// TIA Portal V20 export
// export: Created 2025-12-01T14:57:22.6291622Z, ExportSetting None, DisplayName Totally Integrated Automation Portal, DisplayVersion V20 Update 3, DisplayName TIA Portal Openness, DisplayVersion V20 Update 3, DisplayName TIA Portal Version Control Interface, DisplayVersion V20 Update 3, DisplayName STEP 7 Professional, DisplayVersion V20 Update 3, DisplayName STEP 7 Safety, DisplayVersion V20 Update 2, DisplayName WinCC Basic/Comfort/Advanced, DisplayVersion V20 Update 3, DisplayName WinCC Professional, DisplayVersion V20 Update 3, DisplayName WinCC Unified, DisplayVersion V20 Update 3
FUNCTION "FC1_Llamadas_CCPIF" : Void   // FC1, LAD
{ S7_Optimized_Access := 'FALSE' }
// stored: AutoNumber false, SetENOAutomatically false
   VAR_TEMP
      FinReset : Bool;
      Luminoso_Verde : Bool;
      Luminoso_Rojo : Bool;
      Luminoso_Naranja : Bool;
   END_VAR
BEGIN

REGION Network 1: Final de Reset
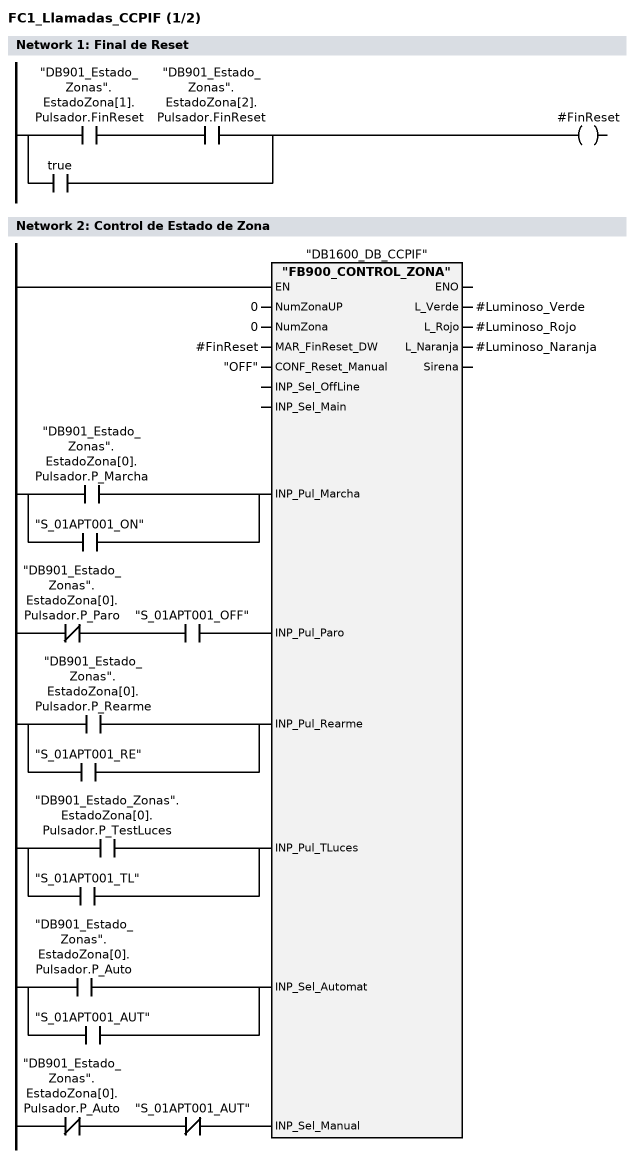
   RUNG wire#powerrail
      Contact( "DB901_Estado_Zonas".EstadoZona[1].Pulsador.FinReset )
      Contact( "DB901_Estado_Zonas".EstadoZona[2].Pulsador.FinReset )
      wire#w1
      Coil( #FinReset )
   END_RUNG
   RUNG wire#powerrail
      Contact( true )
   END_RUNG wire#w1
   // the same network as SCL:
   #FinReset := ("DB901_Estado_Zonas".EstadoZona[1].Pulsador.FinReset AND "DB901_Estado_Zonas".EstadoZona[2].Pulsador.FinReset) OR true;
END_REGION

REGION Network 2: Control de Estado de Zona
   RUNG wire#powerrail
      "DB1600_DB_CCPIF"(INP_Pul_Marcha := wire#w1, INP_Pul_Paro := wire#w2, INP_Pul_Rearme := wire#w3, INP_Pul_TLuces := wire#w4, INP_Sel_Automat := wire#w5, INP_Sel_Manual := wire#w6, NumZonaUP := 0, NumZona := 0, MAR_FinReset_DW := #FinReset, CONF_Reset_Manual := "OFF", INP_Sel_OffLine :=, INP_Sel_Main :=, L_Verde => #Luminoso_Verde, L_Rojo => #Luminoso_Rojo, L_Naranja => #Luminoso_Naranja, Sirena =>)
   END_RUNG
   RUNG wire#powerrail
      Contact( "DB901_Estado_Zonas".EstadoZona[0].Pulsador.P_Marcha )
   END_RUNG wire#w1
   RUNG wire#powerrail
      Contact( "S_01APT001_ON" )
   END_RUNG wire#w1
   RUNG wire#powerrail
      I_Contact( "DB901_Estado_Zonas".EstadoZona[0].Pulsador.P_Paro )
      Contact( "S_01APT001_OFF" )
   END_RUNG wire#w2
   RUNG wire#powerrail
      Contact( "DB901_Estado_Zonas".EstadoZona[0].Pulsador.P_Rearme )
   END_RUNG wire#w3
   RUNG wire#powerrail
      Contact( "S_01APT001_RE" )
   END_RUNG wire#w3
   RUNG wire#powerrail
      Contact( "DB901_Estado_Zonas".EstadoZona[0].Pulsador.P_TestLuces )
   END_RUNG wire#w4
   RUNG wire#powerrail
      Contact( "S_01APT001_TL" )
   END_RUNG wire#w4
   RUNG wire#powerrail
      Contact( "DB901_Estado_Zonas".EstadoZona[0].Pulsador.P_Auto )
   END_RUNG wire#w5
   RUNG wire#powerrail
      Contact( "S_01APT001_AUT" )
   END_RUNG wire#w5
   RUNG wire#powerrail
      I_Contact( "DB901_Estado_Zonas".EstadoZona[0].Pulsador.P_Auto )
      I_Contact( "S_01APT001_AUT" )
   END_RUNG wire#w6
   // the same network as SCL:
   "DB1600_DB_CCPIF"(NumZonaUP := 0,   // "FB900_CONTROL_ZONA"
                     NumZona := 0,
                     MAR_FinReset_DW := #FinReset,
                     CONF_Reset_Manual := "OFF",
                     INP_Pul_Marcha := "DB901_Estado_Zonas".EstadoZona[0].Pulsador.P_Marcha OR "S_01APT001_ON",
                     INP_Pul_Paro := NOT "DB901_Estado_Zonas".EstadoZona[0].Pulsador.P_Paro AND "S_01APT001_OFF",
                     INP_Pul_Rearme := "DB901_Estado_Zonas".EstadoZona[0].Pulsador.P_Rearme OR "S_01APT001_RE",
                     INP_Pul_TLuces := "DB901_Estado_Zonas".EstadoZona[0].Pulsador.P_TestLuces OR "S_01APT001_TL",
                     INP_Sel_Automat := "DB901_Estado_Zonas".EstadoZona[0].Pulsador.P_Auto OR "S_01APT001_AUT",
                     INP_Sel_Manual := NOT "DB901_Estado_Zonas".EstadoZona[0].Pulsador.P_Auto AND NOT "S_01APT001_AUT",
                     L_Verde => #Luminoso_Verde,
                     L_Rojo => #Luminoso_Rojo,
                     L_Naranja => #Luminoso_Naranja);
END_REGION

REGION Network 3: ACTUALIZACION AL SISTEMA ANTIGUO DEL JDT
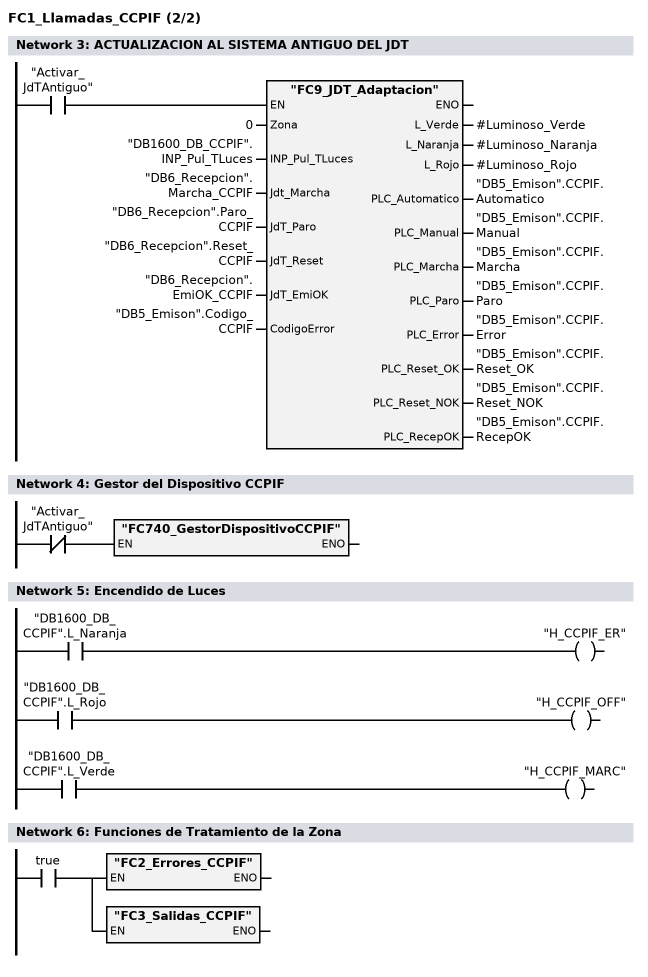
   RUNG wire#powerrail
      Contact( "Activar_JdTAntiguo" )
      "FC9_JDT_Adaptacion"(Zona := 0, INP_Pul_TLuces := "DB1600_DB_CCPIF".INP_Pul_TLuces, Jdt_Marcha := "DB6_Recepcion".Marcha_CCPIF, JdT_Paro := "DB6_Recepcion".Paro_CCPIF, JdT_Reset := "DB6_Recepcion".Reset_CCPIF, JdT_EmiOK := "DB6_Recepcion".EmiOK_CCPIF, CodigoError := "DB5_Emison".Codigo_CCPIF, L_Verde => #Luminoso_Verde, L_Naranja => #Luminoso_Naranja, L_Rojo => #Luminoso_Rojo, PLC_Automatico => "DB5_Emison".CCPIF.Automatico, PLC_Manual => "DB5_Emison".CCPIF.Manual, PLC_Marcha => "DB5_Emison".CCPIF.Marcha, PLC_Paro => "DB5_Emison".CCPIF.Paro, PLC_Error => "DB5_Emison".CCPIF.Error, PLC_Reset_OK => "DB5_Emison".CCPIF.Reset_OK, PLC_Reset_NOK => "DB5_Emison".CCPIF.Reset_NOK, PLC_RecepOK => "DB5_Emison".CCPIF.RecepOK)
   END_RUNG
   // the same network as SCL:
   IF "Activar_JdTAntiguo" THEN
       "FC9_JDT_Adaptacion"(Zona := 0,
                            INP_Pul_TLuces := "DB1600_DB_CCPIF".INP_Pul_TLuces,
                            Jdt_Marcha := "DB6_Recepcion".Marcha_CCPIF,
                            JdT_Paro := "DB6_Recepcion".Paro_CCPIF,
                            JdT_Reset := "DB6_Recepcion".Reset_CCPIF,
                            JdT_EmiOK := "DB6_Recepcion".EmiOK_CCPIF,
                            CodigoError := "DB5_Emison".Codigo_CCPIF,
                            L_Verde => #Luminoso_Verde,
                            L_Naranja => #Luminoso_Naranja,
                            L_Rojo => #Luminoso_Rojo,
                            PLC_Automatico => "DB5_Emison".CCPIF.Automatico,
                            PLC_Manual => "DB5_Emison".CCPIF.Manual,
                            PLC_Marcha => "DB5_Emison".CCPIF.Marcha,
                            PLC_Paro => "DB5_Emison".CCPIF.Paro,
                            PLC_Error => "DB5_Emison".CCPIF.Error,
                            PLC_Reset_OK => "DB5_Emison".CCPIF.Reset_OK,
                            PLC_Reset_NOK => "DB5_Emison".CCPIF.Reset_NOK,
                            PLC_RecepOK => "DB5_Emison".CCPIF.RecepOK);
   END_IF;
END_REGION

REGION Network 4: Gestor del Dispositivo CCPIF
   RUNG wire#powerrail
      I_Contact( "Activar_JdTAntiguo" )
      "FC740_GestorDispositivoCCPIF"()
   END_RUNG
   // the same network as SCL:
   IF NOT "Activar_JdTAntiguo" THEN "FC740_GestorDispositivoCCPIF"(); END_IF;
END_REGION

REGION Network 5: Encendido de Luces
   RUNG wire#powerrail
      Contact( "DB1600_DB_CCPIF".L_Naranja )
      Coil( "H_CCPIF_ER" )
   END_RUNG
   RUNG wire#powerrail
      Contact( "DB1600_DB_CCPIF".L_Rojo )
      Coil( "H_CCPIF_OFF" )
   END_RUNG
   RUNG wire#powerrail
      Contact( "DB1600_DB_CCPIF".L_Verde )
      Coil( "H_CCPIF_MARC" )
   END_RUNG
   // the same network as SCL:
   "H_CCPIF_ER" := "DB1600_DB_CCPIF".L_Naranja;
   "H_CCPIF_OFF" := "DB1600_DB_CCPIF".L_Rojo;
   "H_CCPIF_MARC" := "DB1600_DB_CCPIF".L_Verde;
END_REGION

REGION Network 6: Funciones de Tratamiento de la Zona
   RUNG wire#powerrail
      Contact( true )
      wire#w1
      "FC2_Errores_CCPIF"()
   END_RUNG
   RUNG wire#w1
      "FC3_Salidas_CCPIF"()
   END_RUNG
   // the same network as SCL:
   IF true THEN
       "FC2_Errores_CCPIF"();
       "FC3_Salidas_CCPIF"();
   END_IF;
END_REGION
END_FUNCTION
